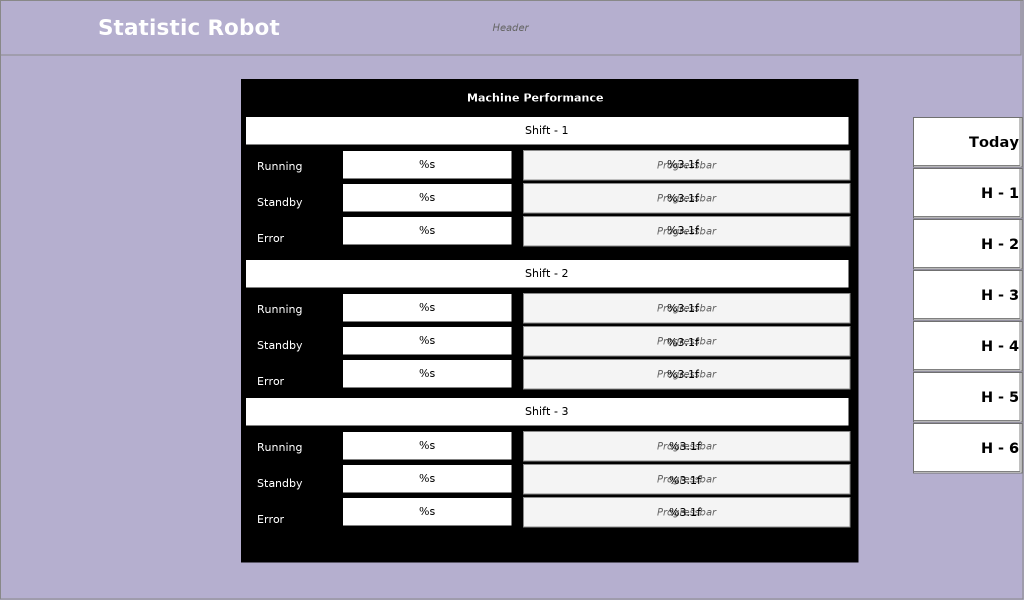
VISUALIZATION OEE_Robot  // 1024x600
    Frame (0,0 1021x55)
        shows Header()
    RoundedRectangle (241,79 617x483)
    RoundedRectangle (245,116 604x29), "Shift - 1"
    Label (268,78 535x40), "Machine Performance"
    Label (254,149 78x35), "Running"
    Label (254,185 78x35), "Standby"
    Label (254,221 78x35), "Error"
    Progressbar (523,150 327x30), variable: Data_GVL.dt_OEETime.Precentage[0].Running
    Progressbar (523,183 327x30), variable: Data_GVL.dt_OEETime.Precentage[0].Stopped
    Progressbar (523,216 327x30), variable: Data_GVL.dt_OEETime.Precentage[0].Error
    RoundedRectangle (342,150 170x29), "%s", text variable: Data_GVL.dt_OEETime.HMI_Time[0].sRunning
    RoundedRectangle (342,183 170x29), "%s", text variable: Data_GVL.dt_OEETime.HMI_Time[0].sStopped
    RoundedRectangle (342,216 170x29), "%s", text variable: Data_GVL.dt_OEETime.HMI_Time[0].sError
    RoundedRectangle (245,259 604x29), "Shift - 2"
    Label (254,292 78x35), "Running"
    Label (254,328 78x35), "Standby"
    Label (254,364 78x35), "Error"
    Progressbar (523,293 327x30), variable: Data_GVL.dt_OEETime.Precentage[1].Running
    Progressbar (523,326 327x30), variable: Data_GVL.dt_OEETime.Precentage[1].Stopped
    Progressbar (523,359 327x30), variable: Data_GVL.dt_OEETime.Precentage[1].Error
    RoundedRectangle (342,293 170x29), "%s", text variable: Data_GVL.dt_OEETime.HMI_Time[1].sRunning
    RoundedRectangle (342,326 170x29), "%s", text variable: Data_GVL.dt_OEETime.HMI_Time[1].sStopped
    RoundedRectangle (342,359 170x29), "%s", text variable: Data_GVL.dt_OEETime.HMI_Time[1].sError
    RoundedRectangle (245,397 604x29), "Shift - 3"
    Label (254,430 78x35), "Running"
    Label (254,466 78x35), "Standby"
    Label (254,502 78x35), "Error"
    Progressbar (523,431 327x30), variable: Data_GVL.dt_OEETime.Precentage[2].Running
    Progressbar (523,464 327x30), variable: Data_GVL.dt_OEETime.Precentage[2].Stopped
    Progressbar (523,497 327x30), variable: Data_GVL.dt_OEETime.Precentage[2].Error
    RoundedRectangle (342,431 170x29), "%s", text variable: Data_GVL.dt_OEETime.HMI_Time[2].sRunning
    RoundedRectangle (342,464 170x29), "%s", text variable: Data_GVL.dt_OEETime.HMI_Time[2].sStopped
    RoundedRectangle (342,497 170x29), "%s", text variable: Data_GVL.dt_OEETime.HMI_Time[2].sError
    Button (913,117 109x50), "Today", image: VisuSymbols.Symbols.CalenderDay
        OnMouseClick: execute { Data_GVL.dt_OEETime.HMI_NumberPrev := 0; }
    Button (913,168 109x50), "H - 1", image: VisuSymbols.Symbols.CalenderDay
        OnMouseClick: execute { Data_GVL.dt_OEETime.HMI_NumberPrev := 1; }
    Button (913,219 109x50), "H - 2", image: VisuSymbols.Symbols.CalenderDay
        OnMouseClick: execute { Data_GVL.dt_OEETime.HMI_NumberPrev := 2; }
    Button (913,270 109x50), "H - 3", image: VisuSymbols.Symbols.CalenderDay
        OnMouseClick: execute { Data_GVL.dt_OEETime.HMI_NumberPrev := 3; }
    Button (913,321 109x50), "H - 4", image: VisuSymbols.Symbols.CalenderDay
        OnMouseClick: execute { Data_GVL.dt_OEETime.HMI_NumberPrev := 4; }
    Button (913,372 109x50), "H - 5", image: VisuSymbols.Symbols.CalenderDay
        OnMouseClick: execute { Data_GVL.dt_OEETime.HMI_NumberPrev := 5; }
    Button (913,423 109x50), "H - 6", image: VisuSymbols.Symbols.CalenderDay
        OnMouseClick: execute { Data_GVL.dt_OEETime.HMI_NumberPrev := 6; }
    RoundedRectangle (598,150 170x29), "%3.1f", text variable: Data_GVL.dt_OEETime.Precentage[0].Running
    RoundedRectangle (598,184 170x29), "%3.1f", text variable: Data_GVL.dt_OEETime.Precentage[0].Stopped
    RoundedRectangle (598,216 170x29), "%3.1f", text variable: Data_GVL.dt_OEETime.Precentage[0].Error
    RoundedRectangle (598,294 170x29), "%3.1f", text variable: Data_GVL.dt_OEETime.Precentage[1].Running
    RoundedRectangle (598,328 170x29), "%3.1f", text variable: Data_GVL.dt_OEETime.Precentage[1].Stopped
    RoundedRectangle (598,360 170x29), "%3.1f", text variable: Data_GVL.dt_OEETime.Precentage[1].Error
    RoundedRectangle (600,432 170x29), "%3.1f", text variable: Data_GVL.dt_OEETime.Precentage[2].Running
    RoundedRectangle (600,466 170x29), "%3.1f", text variable: Data_GVL.dt_OEETime.Precentage[2].Stopped
    RoundedRectangle (600,498 170x29), "%3.1f", text variable: Data_GVL.dt_OEETime.Precentage[2].Error
    Label (95,15 214x25), "Statistic Robot"
END_VISUALIZATION

(* stored: Version 1.1.0.1, ProductVersion 3.1.4024.12
   Visu OEE_Robot: Id {42e97e26-d710-4f1e-9333-04a98f1ac264} *)
